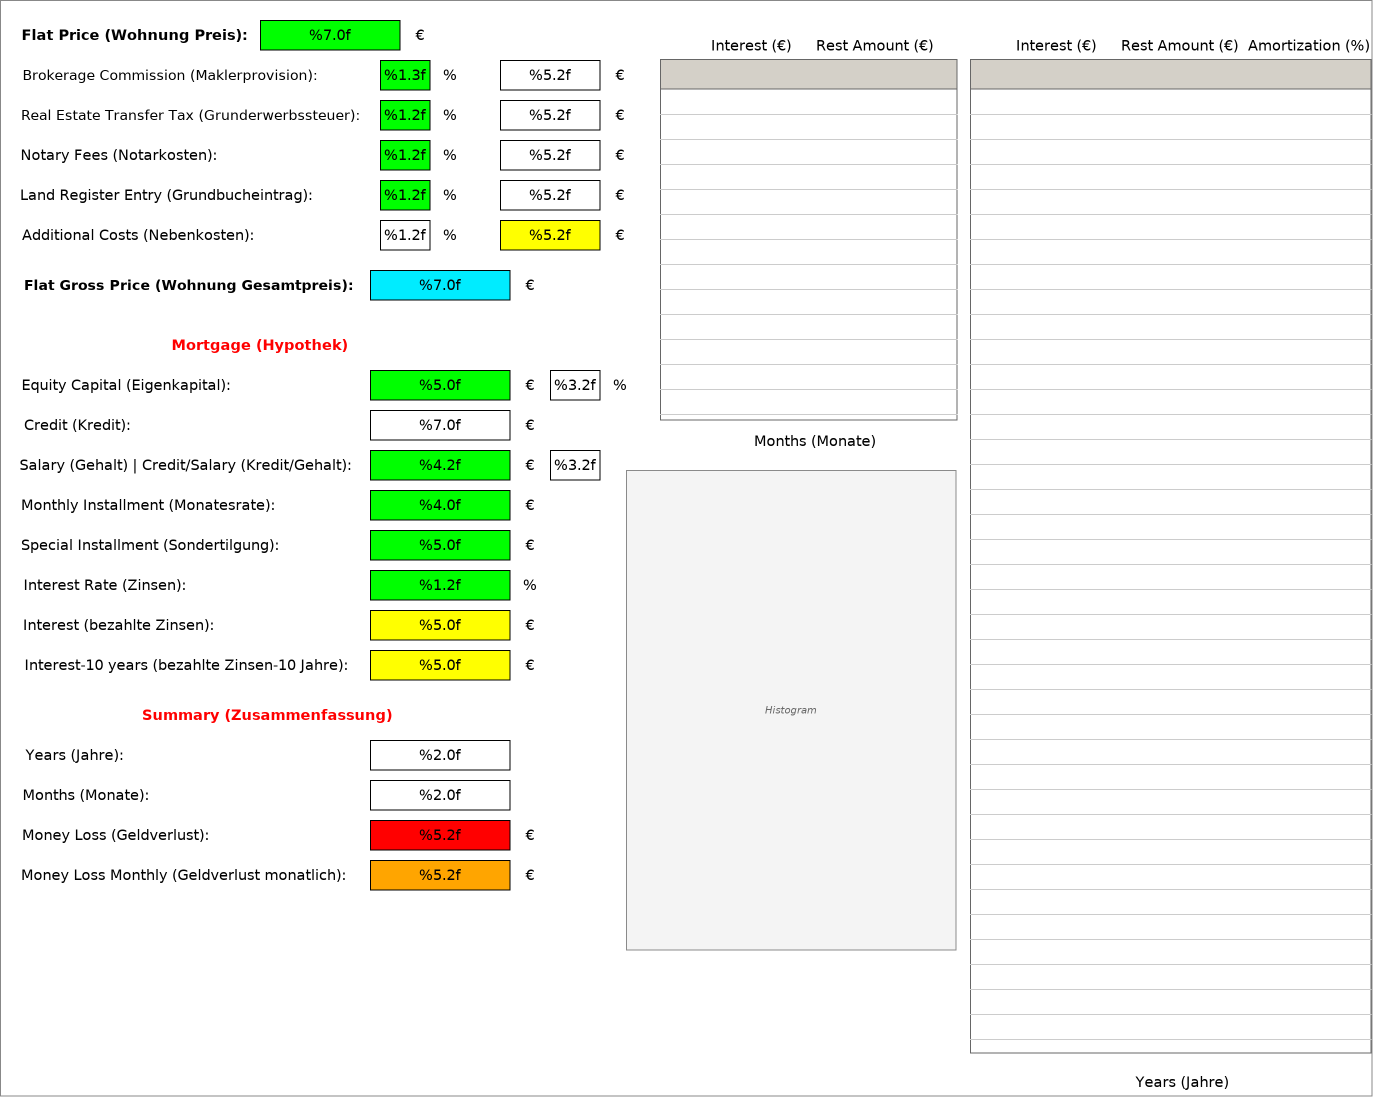
VISUALIZATION Visualization  // 1373x1097
    Textfield (20,20 230x30), "Flat Price (Wohnung Preis):"
    Rectangle (260,20 140x30), "%7.0f", text variable: MAIN.FlatPrice
        OnMouseClick: write the text variable via VisuDialogs.Numpad, min 0, max 1000000
    Rectangle (380,60 50x30), "%1.3f", text variable: MAIN.BrokerageCommissionPercent
        OnMouseClick: write the text variable via VisuDialogs.Numpad, min 0, max 10
    Rectangle (380,100 50x30), "%1.2f", text variable: MAIN.RealEstateTransferTaxPercent
        OnMouseClick: write the text variable via VisuDialogs.Numpad, min 0, max 10
    Rectangle (380,140 50x30), "%1.2f", text variable: MAIN.NotaryFeesPercent
        OnMouseClick: write the text variable via VisuDialogs.Numpad, min 0, max 10
    Rectangle (380,180 50x30), "%1.2f", text variable: MAIN.LandRegisterEntryPercent
        OnMouseClick: write the text variable via VisuDialogs.Numpad, min 0, max 10
    Rectangle (380,220 50x30), "%1.2f", text variable: MAIN.AdditionalCostsPercent
    Textfield (20,60 300x30), "Brokerage Commission (Maklerprovision):"
    Rectangle (500,60 100x30), "%5.2f", text variable: MAIN.BrokerageCommission
    Textfield (20,100 341x30), "Real Estate Transfer Tax (Grunderwerbssteuer):"
    Rectangle (500,100 100x30), "%5.2f", text variable: MAIN.RealEstateTransferTax
    Textfield (20,140 198x30), "Notary Fees (Notarkosten):"
    Rectangle (500,140 100x30), "%5.2f", text variable: MAIN.NotaryFees
    Textfield (20,180 293x30), "Land Register Entry (Grundbucheintrag):"
    Rectangle (500,180 100x30), "%5.2f", text variable: MAIN.LandRegisterEntry
    Textfield (20,220 237x30), "Additional Costs (Nebenkosten):"
    Rectangle (500,220 100x30), "%5.2f", text variable: MAIN.AdditionalCosts
    Textfield (440,60 20x30), "%"
    Textfield (440,100 20x30), "%"
    Textfield (440,140 20x30), "%"
    Textfield (440,180 20x30), "%"
    Textfield (440,220 20x30), "%"
    Textfield (610,60 20x30), "€"
    Textfield (610,100 20x30), "€"
    Textfield (610,140 20x30), "€"
    Textfield (610,180 20x30), "€"
    Textfield (610,220 20x30), "€"
    Textfield (410,20 20x30), "€"
    Textfield (20,270 338x30), "Flat Gross Price (Wohnung Gesamtpreis):"
    Rectangle (370,270 140x30), "%7.0f", text variable: MAIN.FlatGrossPrice
    Textfield (520,270 20x30), "€"
    Textfield (160,330 200x30), "Mortgage (Hypothek)"
    Textfield (20,370 213x30), "Equity Capital (Eigenkapital):"
    Rectangle (370,370 140x30), "%5.0f", text variable: MAIN.Capital
        OnMouseClick: write the text variable via VisuDialogs.Numpad, min 0, max 300000
    Textfield (520,370 20x30), "€"
    Textfield (20,410 115x30), "Credit (Kredit):"
    Rectangle (370,410 140x30), "%7.0f", text variable: MAIN.Credit
    Textfield (520,410 20x30), "€"
    Textfield (20,490 257x30), "Monthly Installment (Monatesrate):"
    Rectangle (370,490 140x30), "%4.0f", text variable: MAIN.MonthlyInstallment
        OnMouseClick: write the text variable via VisuDialogs.Numpad, min 0, max 10000
    Textfield (520,490 20x30), "€"
    Textfield (20,570 170x30), "Interest Rate (Zinsen):"
    Rectangle (370,570 140x30), "%1.2f", text variable: MAIN.InterestRate
        OnMouseClick: write the text variable via VisuDialogs.Numpad, min 0, max 5
    Textfield (520,570 20x30), "%"
    Table (660,59 297x361), data array: MAIN.arVisu
        p3854506369: MAIN.arVisu[1][INDEX]
        p1892666644: MAIN.arVisu[2][INDEX]
    Textfield (20,610 198x30), "Interest (bezahlte Zinsen):"
    Rectangle (370,610 140x30), "%5.0f", text variable: MAIN.PaidInterest
    Textfield (520,610 20x30), "€"
    Table (970,59 401x994), data array: MAIN.arVisu2
        p3854506369: MAIN.arVisu2[1][INDEX]
        p1892666644: MAIN.arVisu2[2][INDEX]
        p338671338: MAIN.arVisu2[3][INDEX]
    Textfield (20,740 110x30), "Years (Jahre):"
    Rectangle (370,740 140x30), "%2.0f", text variable: MAIN.PaymentYears
    Textfield (18,780 136x30), "Months (Monate):"
    Rectangle (370,780 140x30), "%2.0f", text variable: MAIN.PaymentMonths
    Textfield (750,426 130x30), "Months (Monate)"
    Textfield (1135,1067 95x30), "Years (Jahre)"
    Textfield (710,33 83x25), "Interest (€)"
    Textfield (815,33 120x25), "Rest Amount (€)"
    Textfield (1015,33 83x25), "Interest (€)"
    Textfield (1120,33 120x25), "Rest Amount (€)"
    Textfield (140,700 255x30), "Summary (Zusammenfassung)"
    Textfield (20,820 192x30), "Money Loss (Geldverlust):"
    Rectangle (370,820 140x30), "%5.2f", text variable: MAIN.MoneyLoss
    Textfield (520,820 20x30), "€"
    Rectangle (550,370 50x30), "%3.2f", text variable: MAIN.CapitalPercent
    Textfield (610,370 20x30), "%"
    Textfield (20,860 328x30), "Money Loss Monthly (Geldverlust monatlich):"
    Rectangle (370,860 140x30), "%5.2f", text variable: MAIN.MoneyLossMonthly
    Textfield (520,860 20x30), "€"
    Textfield (20,650 333x30), "Interest-10 years (bezahlte Zinsen-10 Jahre):"
    Rectangle (370,650 140x30), "%5.0f", text variable: MAIN.PaidInterest10years
    Textfield (520,650 20x30), "€"
    Textfield (20,450 332x30), "Salary (Gehalt) | Credit/Salary (Kredit/Gehalt):"
    Rectangle (370,450 140x30), "%4.2f", text variable: MAIN.Salary
        OnMouseClick: write the text variable via VisuDialogs.Numpad, min 0, max 150000
    Textfield (520,450 20x30), "€"
    Rectangle (550,450 50x30), "%3.2f", text variable: MAIN.CreditPercent
    Textfield (1245,33 128x25), "Amortization (%)"
    Textfield (20,530 261x30), "Special Installment (Sondertilgung):"
    Rectangle (370,530 140x30), "%5.0f", text variable: MAIN.SpecialInstallment
        OnMouseClick: write the text variable via VisuDialogs.Numpad, min 0, max 25000
    Textfield (520,530 20x30), "€"
    Histogram (626,470 330x480), scale format: %.1f, scale 0..600000
        p1518820177: MAIN.arVisu[2]
        p102497268: MAIN.arVisu[2]
        p788070771: ARRAY [1..(Years * 12)] OF REAL
END_VISUALIZATION

(* stored: Version 1.1.0.1, ProductVersion 3.1.4024.6
   Visu Visualization: Id {8b1dc8e8-b46e-4bea-a45f-955749f5e274} *)
